// TIA Portal V21 export
TYPE "LBC_typeMotorStarterCommands"
TITLE = LBC_typeMotorStarterCommands
// Module related manual commands from HMI
   STRUCT
      refreshConfiguration : Bool;   // Copy global configuration parameters into module interface for external systems
      editConfiguration : Bool;   // Edit mode for configuration parameters in control system is active - copying into module interface is stopped
      saveConfiguration : Bool;   // Save configuration parameters from module interface into to global configuration parameters after change
      reset : Bool;   // Manual reset command from HMI, Reset the motor starter. Output `resetStarter` is TRUE at least for the time configured at parameter `resetTime`
      commandForward : Bool;   // Manual forward command from HMI, Rising edge: Start the motor forward
      commandBackward : Bool;   // Manual backward command from HMI, Rising edge: Start the motor backward
   END_STRUCT;
END_TYPE
